// TIA Portal project "SCADA_TRAFFIC_LAMP" (V15)

(* hardware
DEVICE "PC-System_1"  SIMATIC PC station
   slot 0: "SIMATIC PC station"  Rail  SIMATIC PC-Station  V1.0
      slot 125: "Stationmanager"  Station_Manager  V6.0.4
   slot 1: "HMI_RT_1"  WinCC RT Advanced  6AV2 104-0xxxx-xxxx  15.0.0.0
      slot 33792: "Host interface"  Host interface
   slot 2: "IE general_1"  IE General  IE_CP  V8.2.0
DEVICE "S7-1200 station_1"  S7-1200 Station
   slot 0: "Rack_0"  S7-1200 Rack  Rack  V1.0
   slot 1: "PLC_1"  CPU 1214C AC/DC/Rly  6ES7 214-1BG40-0XB0  V4.2
*)

// ===== PLC "PLC_1"  CPU 1214C AC/DC/Rly =====

VAR_GLOBAL   // PLC tag table "Default tag table"
   "System_Byte" AT %MB1 : Byte;
   "FirstScan" AT %M1.0 : Bool;
   "DiagStatusUpdate" AT %M1.1 : Bool;
   "AlwaysTRUE" AT %M1.2 : Bool;
   "AlwaysFALSE" AT %M1.3 : Bool;
   "Clock_Byte" AT %MB0 : Byte;
   "Clock_10Hz" AT %M0.0 : Bool;
   "Clock_5Hz" AT %M0.1 : Bool;
   "Clock_2.5Hz" AT %M0.2 : Bool;
   "Clock_2Hz" AT %M0.3 : Bool;
   "Clock_1.25Hz" AT %M0.4 : Bool;
   "Clock_1Hz" AT %M0.5 : Bool;
   "Clock_0.625Hz" AT %M0.6 : Bool;
   "Clock_0.5Hz" AT %M0.7 : Bool;
   "On" AT %M2.0 : Bool;
   "Off" AT %M2.1 : Bool;
   "yellow_1" AT %Q0.0 : Bool;
   "green_1" AT %Q0.1 : Bool;
   "red_1" AT %Q0.2 : Bool;
   "yellow_2" AT %Q0.3 : Bool;
   "green_2" AT %Q0.4 : Bool;
   "red_2" AT %Q0.5 : Bool;
   "tg_run_system" AT %Q0.6 : Bool;
   "Set_green_lamp" AT %MW100 : Int;
   "Set_red_lamp" AT %MW102 : Int;
   "Cal_yellow_lamp" AT %MW104 : Int;
   "Sum_time" AT %MW106 : Int;
   "Tag_1" AT %M50.0 : Bool;
   "Time_actual" AT %MW108 : Int;
   "Step1" AT %MW4 : Int;
   "Step2" AT %MW6 : Int;
   "Step3" AT %MW8 : Int;
   "Step4" AT %MW10 : Int;
   "Time_green_1" AT %MW12 : Int;
   "Time_yellow_1" AT %MW14 : Int;
   "Time_red_1" AT %MW16 : Int;
   "Time_green_2" AT %MW18 : Int;
   "Time_yellow_2" AT %MW20 : Int;
   "Time_red_2" AT %MW22 : Int;
END_VAR

ORGANIZATION_BLOCK "Main"   // OB1, LAD, ProgramCycle
TITLE = "Main Program Sweep (Cycle)"
{ S7_Optimized_Access := 'TRUE' }
VERSION : 0.1
   VAR_INPUT
      Initial_Call : Bool;   // Initial call of this OB
      Remanence : Bool;   // =True, if remanent data are available
   END_VAR
   VAR_TEMP   // added for the SCL form of the ladder/FBD networks
      _w1 : Bool;
      _w2 : Bool;
   END_VAR
BEGIN

REGION Network 1
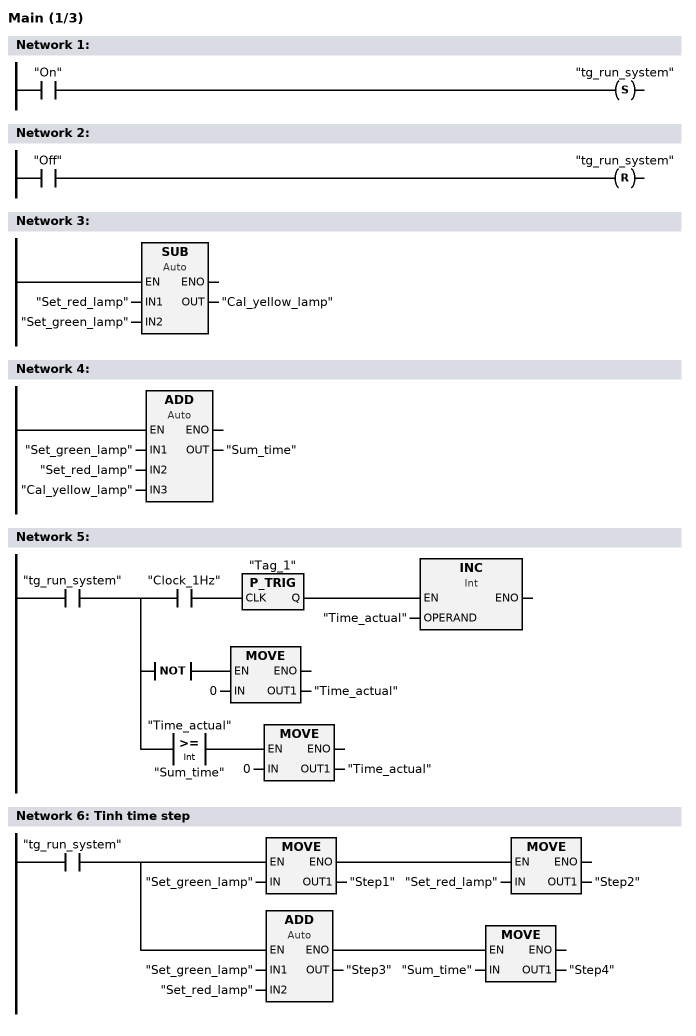
   RUNG wire#powerrail
      Contact( "On" )
      S_Coil( "tg_run_system" )
   END_RUNG
   // the same network as SCL:
   IF "On" THEN "tg_run_system" := TRUE; END_IF;
END_REGION

REGION Network 2
   RUNG wire#powerrail
      Contact( "Off" )
      R_Coil( "tg_run_system" )
   END_RUNG
   // the same network as SCL:
   IF "Off" THEN "tg_run_system" := FALSE; END_IF;
END_REGION

REGION Network 3
   RUNG wire#powerrail
      Sub(in1 := "Set_red_lamp", in2 := "Set_green_lamp", out => "Cal_yellow_lamp")
   END_RUNG
   // the same network as SCL:
   "Cal_yellow_lamp" := "Set_red_lamp" - "Set_green_lamp";
END_REGION

REGION Network 4
   RUNG wire#powerrail
      Add(in1 := "Set_green_lamp", in2 := "Set_red_lamp", in3 := "Cal_yellow_lamp", out => "Sum_time")
   END_RUNG
   // the same network as SCL:
   "Sum_time" := "Set_green_lamp" + "Set_red_lamp" + "Cal_yellow_lamp";
END_REGION

REGION Network 5
   RUNG wire#powerrail
      Contact( "tg_run_system" )
      wire#w1
      Contact( "Clock_1Hz" )
      P_Trig( "Tag_1" )
      { S7_Templates := "DestType := Int" } Inc( "Time_actual" )
   END_RUNG
   RUNG wire#w1
      Not()
      Move(in := 0, out1 => "Time_actual")
   END_RUNG
   RUNG wire#w1
      { S7_Templates := "SrcType := Int" } GE_Contact(in1 := "Time_actual", in2 := "Sum_time")
      Move(in := 0, out1 => "Time_actual")
   END_RUNG
   // the same network as SCL:
   #_w1 := "tg_run_system" AND "Clock_1Hz";
   #_w2 := #_w1 AND NOT "Tag_1";   // rising edge
   "Tag_1" := #_w1;
   IF #_w2 THEN "Time_actual" := "Time_actual" + 1; END_IF;
   IF NOT "tg_run_system" THEN "Time_actual" := 0; END_IF;
   IF "tg_run_system" AND ("Time_actual" >= "Sum_time") THEN "Time_actual" := 0; END_IF;
END_REGION

REGION Network 6: Tinh time step
   RUNG wire#powerrail
      Contact( "tg_run_system" )
      wire#w1
      Move(in := "Set_green_lamp", out1 => "Step1")
      Move(in := "Set_red_lamp", out1 => "Step2")
   END_RUNG
   RUNG wire#w1
      Add(in1 := "Set_green_lamp", in2 := "Set_red_lamp", out => "Step3")
      Move(in := "Sum_time", out1 => "Step4")
   END_RUNG
   // the same network as SCL:
   IF "tg_run_system" THEN
       "Step1" := "Set_green_lamp";
       "Step2" := "Set_red_lamp";
       "Step3" := "Set_green_lamp" + "Set_red_lamp";
       "Step4" := "Sum_time";
   END_IF;
END_REGION

REGION Network 7: A
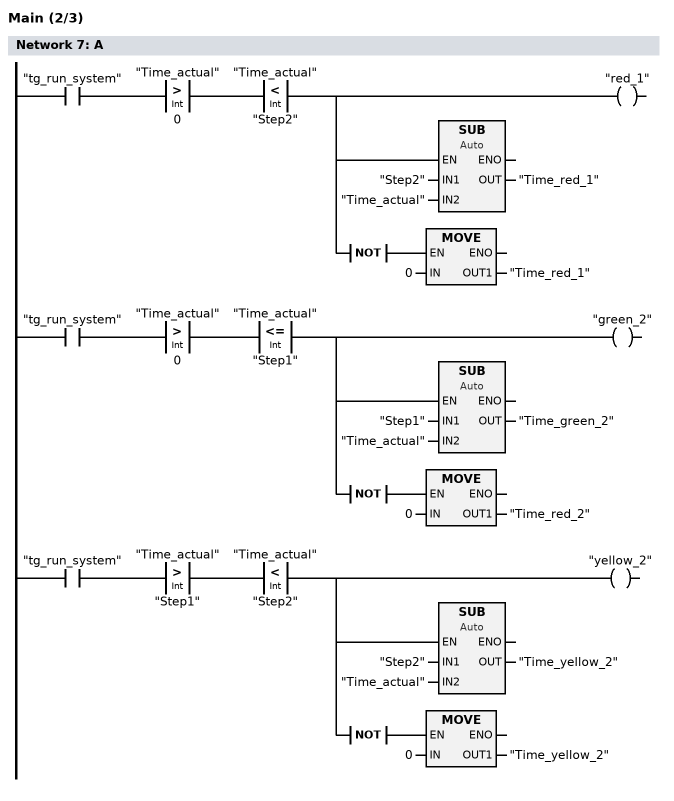
   RUNG wire#powerrail
      Contact( "tg_run_system" )
      { S7_Templates := "SrcType := Int" } GT_Contact(in1 := "Time_actual", in2 := 0)
      { S7_Templates := "SrcType := Int" } LT_Contact(in1 := "Time_actual", in2 := "Step2")
      wire#w1
      Coil( "red_1" )
   END_RUNG
   RUNG wire#w1
      Sub(in1 := "Step2", in2 := "Time_actual", out => "Time_red_1")
   END_RUNG
   RUNG wire#w1
      Not()
      Move(in := 0, out1 => "Time_red_1")
   END_RUNG
   RUNG wire#powerrail
      Contact( "tg_run_system" )
      { S7_Templates := "SrcType := Int" } GT_Contact(in1 := "Time_actual", in2 := 0)
      { S7_Templates := "SrcType := Int" } LE_Contact(in1 := "Time_actual", in2 := "Step1")
      wire#w2
      Coil( "green_2" )
   END_RUNG
   RUNG wire#w2
      Sub(in1 := "Step1", in2 := "Time_actual", out => "Time_green_2")
   END_RUNG
   RUNG wire#w2
      Not()
      Move(in := 0, out1 => "Time_red_2")
   END_RUNG
   RUNG wire#powerrail
      Contact( "tg_run_system" )
      { S7_Templates := "SrcType := Int" } GT_Contact(in1 := "Time_actual", in2 := "Step1")
      { S7_Templates := "SrcType := Int" } LT_Contact(in1 := "Time_actual", in2 := "Step2")
      wire#w3
      Coil( "yellow_2" )
   END_RUNG
   RUNG wire#w3
      Sub(in1 := "Step2", in2 := "Time_actual", out => "Time_yellow_2")
   END_RUNG
   RUNG wire#w3
      Not()
      Move(in := 0, out1 => "Time_yellow_2")
   END_RUNG
   // the same network as SCL:
   "red_1" := "tg_run_system" AND ("Time_actual" > 0) AND ("Time_actual" < "Step2");
   IF "red_1" THEN "Time_red_1" := "Step2" - "Time_actual"; END_IF;
   IF NOT "red_1" THEN "Time_red_1" := 0; END_IF;
   "green_2" := "tg_run_system" AND ("Time_actual" > 0) AND ("Time_actual" <= "Step1");
   IF "green_2" THEN "Time_green_2" := "Step1" - "Time_actual"; END_IF;
   IF NOT "green_2" THEN "Time_red_2" := 0; END_IF;
   "yellow_2" := "tg_run_system" AND ("Time_actual" > "Step1") AND ("Time_actual" < "Step2");
   IF "yellow_2" THEN "Time_yellow_2" := "Step2" - "Time_actual"; END_IF;
   IF NOT "yellow_2" THEN "Time_yellow_2" := 0; END_IF;
END_REGION

REGION Network 8: B
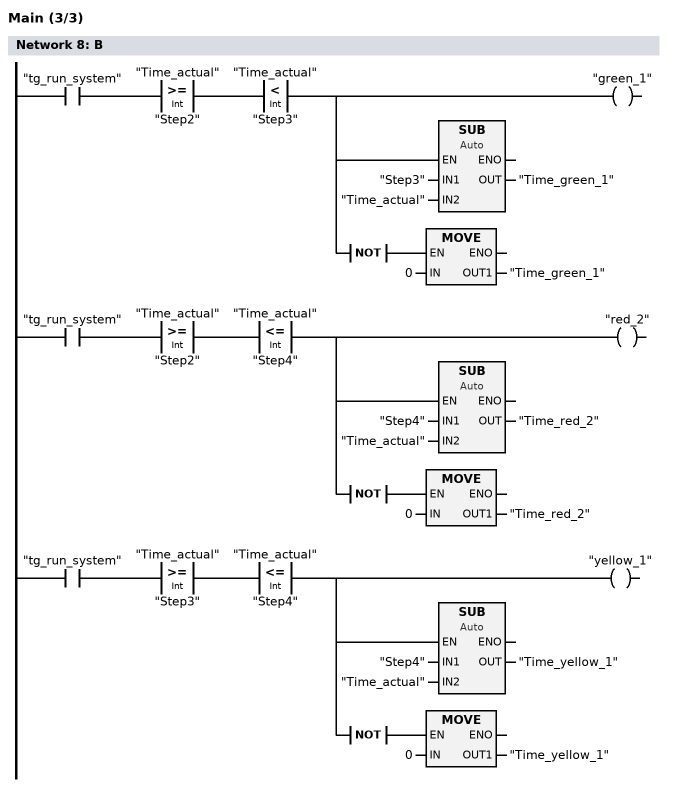
   RUNG wire#powerrail
      Contact( "tg_run_system" )
      { S7_Templates := "SrcType := Int" } GE_Contact(in1 := "Time_actual", in2 := "Step2")
      { S7_Templates := "SrcType := Int" } LT_Contact(in1 := "Time_actual", in2 := "Step3")
      wire#w1
      Coil( "green_1" )
   END_RUNG
   RUNG wire#w1
      Sub(in1 := "Step3", in2 := "Time_actual", out => "Time_green_1")
   END_RUNG
   RUNG wire#w1
      Not()
      Move(in := 0, out1 => "Time_green_1")
   END_RUNG
   RUNG wire#powerrail
      Contact( "tg_run_system" )
      { S7_Templates := "SrcType := Int" } GE_Contact(in1 := "Time_actual", in2 := "Step2")
      { S7_Templates := "SrcType := Int" } LE_Contact(in1 := "Time_actual", in2 := "Step4")
      wire#w2
      Coil( "red_2" )
   END_RUNG
   RUNG wire#w2
      Sub(in1 := "Step4", in2 := "Time_actual", out => "Time_red_2")
   END_RUNG
   RUNG wire#w2
      Not()
      Move(in := 0, out1 => "Time_red_2")
   END_RUNG
   RUNG wire#powerrail
      Contact( "tg_run_system" )
      { S7_Templates := "SrcType := Int" } GE_Contact(in1 := "Time_actual", in2 := "Step3")
      { S7_Templates := "SrcType := Int" } LE_Contact(in1 := "Time_actual", in2 := "Step4")
      wire#w3
      Coil( "yellow_1" )
   END_RUNG
   RUNG wire#w3
      Sub(in1 := "Step4", in2 := "Time_actual", out => "Time_yellow_1")
   END_RUNG
   RUNG wire#w3
      Not()
      Move(in := 0, out1 => "Time_yellow_1")
   END_RUNG
   // the same network as SCL:
   "green_1" := "tg_run_system" AND ("Time_actual" >= "Step2") AND ("Time_actual" < "Step3");
   IF "green_1" THEN "Time_green_1" := "Step3" - "Time_actual"; END_IF;
   IF NOT "green_1" THEN "Time_green_1" := 0; END_IF;
   "red_2" := "tg_run_system" AND ("Time_actual" >= "Step2") AND ("Time_actual" <= "Step4");
   IF "red_2" THEN "Time_red_2" := "Step4" - "Time_actual"; END_IF;
   IF NOT "red_2" THEN "Time_red_2" := 0; END_IF;
   "yellow_1" := "tg_run_system" AND ("Time_actual" >= "Step3") AND ("Time_actual" <= "Step4");
   IF "yellow_1" THEN "Time_yellow_1" := "Step4" - "Time_actual"; END_IF;
   IF NOT "yellow_1" THEN "Time_yellow_1" := 0; END_IF;
END_REGION
END_ORGANIZATION_BLOCK

ORGANIZATION_BLOCK "Startup"   // OB100, LAD, Startup
TITLE = "Complete Restart"
{ S7_Optimized_Access := 'TRUE' }
VERSION : 0.1
   VAR_INPUT
      LostRetentive : Bool;   // True if retentive data are lost
      LostRTC : Bool;   // True if date and time are lost
   END_VAR
BEGIN

REGION Network 1
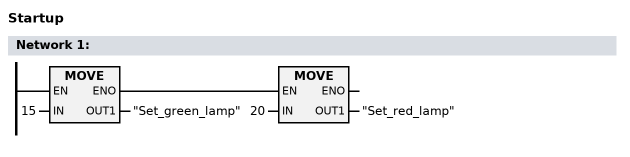
   RUNG wire#powerrail
      Move(in := 15, out1 => "Set_green_lamp")
      Move(in := 20, out1 => "Set_red_lamp")
   END_RUNG
   // the same network as SCL:
   "Set_green_lamp" := 15;
   "Set_red_lamp" := 20;
END_REGION
END_ORGANIZATION_BLOCK

(* ===== HMI "HMI_RT_1" =====
system functions are stored by id; their names below are inferred from use
connection "HMI_Connection_1": ETHERNET, S7_1200_OMS

HMI tags "Default tag table"
   "On" : Bool = PLC On AT %M2.0, 1 s
   "Off" : Bool = PLC Off AT %M2.1, 1 s
   "tg_run_system" : Bool = PLC tg_run_system AT %Q0.6, 1 s
   "Set_green_lamp" : Int = PLC Set_green_lamp AT %MW100, 1 s
   "Set_red_lamp" : Int = PLC Set_red_lamp AT %MW102, 1 s
   "green_1" : Bool = PLC green_1 AT %Q0.1, 1 s
   "yellow_1" : Bool = PLC yellow_1 AT %Q0.0, 1 s
   "red_1" : Bool = PLC red_1 AT %Q0.2, 1 s
   "green_2" : Bool = PLC green_2 AT %Q0.4, 1 s
   "Time_yellow_2" : Int = PLC Time_yellow_2 AT %MW20, 1 s
   "yellow_2" : Bool = PLC yellow_2 AT %Q0.3, 1 s
   "red_2" : Bool = PLC red_2 AT %Q0.5, 1 s
   "Time_green_1" : Int = PLC Time_green_1 AT %MW12, 1 s
   "Time_yellow_1" : Int = PLC Time_yellow_1 AT %MW14, 1 s
   "Time_red_1" : Int = PLC Time_red_1 AT %MW16, 1 s
   "Time_green_2" : Int = PLC Time_green_2 AT %MW18, 1 s
   "Time_red_2" : Int = PLC Time_red_2 AT %MW22, 1 s

screen "Screen_1" 1024x768
   TextField "Text field_1" at 430,11 size 154x34; Text 'Traffic_lamp'
   TextField "Text field_2" at 649,328 size 20x32; Text '1'
   TextField "Text field_3" at 325,326 size 20x32; Text '1'
   TextField "Text field_4" at 498,158 size 20x32; Text '2'
   TextField "Text field_5" at 493,480 size 20x32; Text '2'
   Circle "Circle_1" at 583,223 size 48x48
      Appearance <- "green_2"
   Circle "Circle_2" at 650,223 size 48x48
      Appearance <- "yellow_2"
   Circle "Circle_3" at 713,224 size 48x48
      Appearance <- "red_2"
   Circle "Circle_7" at 584,421 size 48x48
      Appearance <- "green_1"
   Circle "Circle_8" at 584,474 size 48x48
      Appearance <- "yellow_1"
   Circle "Circle_9" at 584,528 size 48x48
      Appearance <- "red_1"
   Button "Button_1" at 721,35 size 75x54; TextOff 'ON'
      on Press: SetBit("On")
      on Release: ResetBit("On")
   Button "Button_2" at 721,104 size 75x54; TextOff 'OFF'
      on Press: SetBit("Off")
      on Release: ResetBit("Off")
   Circle "Circle_13" at 820,64 size 64x64
      Appearance <- "tg_run_system"
   TextField "Text field_6" at 831,130 size 123x27; Text 'Run_system'
   IOField "I/O field_1" at 141,73 size 96x48; FormatPattern 99999; Unit  s
      Appearance <- "Set_green_lamp"
      ProcessValue <- "Set_green_lamp"
   TextField "Text field_7" at 4,73 size 114x29; Text 'Set_Green'
   IOField "I/O field_2" at 141,135 size 96x47; FormatPattern 99999; Unit  s
      ProcessValue <- "Set_red_lamp"
   TextField "Text field_8" at 18,142 size 92x29; Text 'Set_Red'
   IOField "I/O field_3" at 750,419 size 96x32; FormatPattern 99999; Unit  s
      ProcessValue <- "Time_green_1"
   IOField "I/O field_4" at 750,475 size 96x32; FormatPattern 99999; Unit  s
      ProcessValue <- "Time_yellow_1"
   IOField "I/O field_5" at 750,526 size 96x32; FormatPattern 99999; Unit  s
      ProcessValue <- "Time_red_1"
   TextField "Text field_9" at 644,425 size 59x21; Text 'green 1'
   TextField "Text field_10" at 643,484 size 62x21; Text 'yellow 1'
   TextField "Text field_11" at 657,544 size 39x21; Text 'red 1'
   Circle "Circle_14" at 383,118 size 48x48
      Appearance <- "green_1"
   Circle "Circle_15" at 383,171 size 48x48
      Appearance <- "yellow_1"
   Circle "Circle_16" at 383,225 size 48x48
      Appearance <- "red_1"
   Circle "Circle_4" at 387,417 size 48x48
      Appearance <- "green_2"
   Circle "Circle_5" at 328,415 size 48x48
      Appearance <- "yellow_2"
   Circle "Circle_6" at 268,416 size 48x48
      Appearance <- "red_2"
   IOField "I/O field_6" at 139,424 size 96x32; FormatPattern 99999; Unit  s
      ProcessValue <- "Time_green_2"
   IOField "I/O field_7" at 139,480 size 96x32; FormatPattern 99999; Unit  s
      ProcessValue <- "Time_yellow_2"
   IOField "I/O field_8" at 139,531 size 96x32; FormatPattern 99999; Unit  s
      ProcessValue <- "Time_red_2"
   TextField "Text field_12" at 51,433 size 64x23; Text 'green 2'
   TextField "Text field_13" at 50,489 size 72x23; Text 'yellow 2'
   TextField "Text field_14" at 79,541 size 43x23; Text 'red 2'
*)